Fanuc KAREL source: IO0030.KL

-- PROVISIONAL review KL for V940-1; original PC SHA256 f944be26d03f428506b4783b926b0f9f10eaaa949c185416fea87cde0a54b9c9
-- Incomplete behavior may be omitted. Consult companion uncertainty JSON. Do not deploy.
PROGRAM IO0030
%NOLOCKGROUP
-- UNRESOLVED_LOCAL_POOL 5 cells at code offset 13; source declarations unknown
-- DIRECT_LOCAL_WORD_ACCESS alone does not prove INTEGER, REAL, or BOOLEAN
BEGIN
  -- V9_ZERO_TABLE_METADATA_HINT layout=0001; no indexed target words; source/name/runtime held
  -- V9_ZERO_GLOBAL_LAYOUT_HINT count-one $GROUP table, zero relocation slots, two routine descriptors; executable preamble and source held
  -- UNRESOLVED_PC offsets 0-18; opcodes 2B,2C,7B
  -- UNRESOLVED_PC offsets 23-30; opcodes 9D,23
  -- UNRESOLVED_PC offsets 35-49; opcodes 2E,22,9D,33,35
  -- UNRESOLVED_PC offsets 54-61; opcodes 9D,23
  -- UNRESOLVED_PC offsets 66-77; opcodes 2E,23
  -- UNRESOLVED_PC offsets 82-98; opcodes 21,21,9D,52,1A
  -- UNRESOLVED_PC offsets 103-107; opcodes 7F
  -- UNRESOLVED_PC offsets 112-116; opcodes 27,AA
  -- UNRESOLVED_PC offsets 121-125; opcodes 7F
END IO0030
